// TIA Portal V16 export
// export: Created 2023-09-11T12:14:53.3184861Z, ExportSetting WithDefaults, DisplayName Totally Integrated Automation Portal, DisplayVersion V16 Update 6, DisplayName TIA Portal Version Control Interface, DisplayVersion V16 Update 2, DisplayName TIA Portal Openness, DisplayVersion V16 Update 6, DisplayName STEP 7 Professional, DisplayVersion V16 Update 6, DisplayName STEP 7 Safety, DisplayVersion V16, DisplayName WinCC Advanced, DisplayVersion V16 Update 6
FUNCTION "01_E_alarm handling" : Void   // FC10, LAD
TITLE = Boks Ready
{ S7_Optimized_Access := 'TRUE' }
AUTHOR : R.Tecmer
VERSION : 0.1
// Handling of alarms. Signaling and deleting
// stored: AutoNumber true, IsIECCheckEnabled false, SetENOAutomatically false, UDAEnableTagReadback false
   VAR_TEMP   // added for the SCL form of the ladder/FBD networks
      _w1 : Bool;
   END_VAR
BEGIN

REGION Network 1: Ready Inverters No1 No2
   // połączyłem bo usunięto drugi falownik
   // Jeśli brak gotowości to ustaw bity
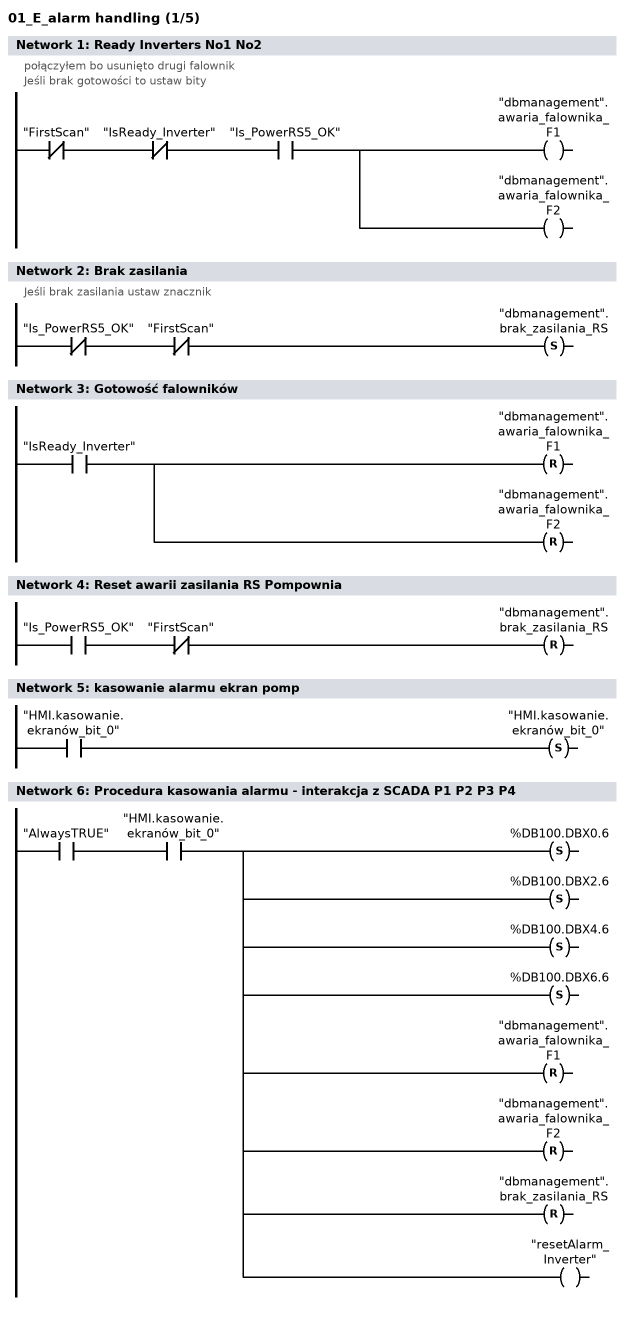
   RUNG wire#powerrail
      I_Contact( "FirstScan" )
      I_Contact( "IsReady_Inverter" )
      Contact( "Is_PowerRS5_OK" )
      wire#w1
      Coil( "dbmanagement".awaria_falownika_F1 )
   END_RUNG
   RUNG wire#w1
      Coil( "dbmanagement".awaria_falownika_F2 )
   END_RUNG
   // the same network as SCL:
   "dbmanagement".awaria_falownika_F1 := NOT "FirstScan" AND NOT "IsReady_Inverter" AND "Is_PowerRS5_OK";
   "dbmanagement".awaria_falownika_F2 := "dbmanagement".awaria_falownika_F1;
END_REGION

REGION Network 2: Brak zasilania
   // Jeśli brak zasilania ustaw znacznik
   RUNG wire#powerrail
      I_Contact( "Is_PowerRS5_OK" )
      I_Contact( "FirstScan" )
      S_Coil( "dbmanagement".brak_zasilania_RS )
   END_RUNG
   // the same network as SCL:
   IF NOT "Is_PowerRS5_OK" AND NOT "FirstScan" THEN "dbmanagement".brak_zasilania_RS := TRUE; END_IF;
END_REGION

REGION Network 3: Gotowość falowników
   RUNG wire#powerrail
      Contact( "IsReady_Inverter" )
      wire#w1
      R_Coil( "dbmanagement".awaria_falownika_F1 )
   END_RUNG
   RUNG wire#w1
      R_Coil( "dbmanagement".awaria_falownika_F2 )
   END_RUNG
   // the same network as SCL:
   IF "IsReady_Inverter" THEN
       "dbmanagement".awaria_falownika_F1 := FALSE;
       "dbmanagement".awaria_falownika_F2 := FALSE;
   END_IF;
END_REGION

REGION Network 4: Reset awarii zasilania RS Pompownia
   RUNG wire#powerrail
      Contact( "Is_PowerRS5_OK" )
      I_Contact( "FirstScan" )
      R_Coil( "dbmanagement".brak_zasilania_RS )
   END_RUNG
   // the same network as SCL:
   IF "Is_PowerRS5_OK" AND NOT "FirstScan" THEN "dbmanagement".brak_zasilania_RS := FALSE; END_IF;
END_REGION

REGION Network 5: kasowanie alarmu ekran pomp
   RUNG wire#powerrail
      Contact( "HMI.kasowanie.ekranów_bit_0" )
      S_Coil( "HMI.kasowanie.ekranów_bit_0" )
   END_RUNG
   // the same network as SCL:
   IF "HMI.kasowanie.ekranów_bit_0" THEN "HMI.kasowanie.ekranów_bit_0" := TRUE; END_IF;
END_REGION

REGION Network 6: Procedura kasowania alarmu - interakcja z SCADA P1 P2 P3 P4
   RUNG wire#powerrail
      Contact( "AlwaysTRUE" )
      Contact( "HMI.kasowanie.ekranów_bit_0" )
      wire#w1
      S_Coil( %DB100.DBX0.6 )
   END_RUNG
   RUNG wire#w1
      S_Coil( %DB100.DBX2.6 )
   END_RUNG
   RUNG wire#w1
      S_Coil( %DB100.DBX4.6 )
   END_RUNG
   RUNG wire#w1
      S_Coil( %DB100.DBX6.6 )
   END_RUNG
   RUNG wire#w1
      R_Coil( "dbmanagement".awaria_falownika_F1 )
   END_RUNG
   RUNG wire#w1
      R_Coil( "dbmanagement".awaria_falownika_F2 )
   END_RUNG
   RUNG wire#w1
      R_Coil( "dbmanagement".brak_zasilania_RS )
   END_RUNG
   RUNG wire#w1
      Coil( "resetAlarm_Inverter" )
   END_RUNG
   // the same network as SCL:
   #_w1 := "AlwaysTRUE" AND "HMI.kasowanie.ekranów_bit_0";
   IF #_w1 THEN
       %DB100.DBX0.6 := TRUE;
       %DB100.DBX2.6 := TRUE;
       %DB100.DBX4.6 := TRUE;
       %DB100.DBX6.6 := TRUE;
       "dbmanagement".awaria_falownika_F1 := FALSE;
       "dbmanagement".awaria_falownika_F2 := FALSE;
       "dbmanagement".brak_zasilania_RS := FALSE;
   END_IF;
   "resetAlarm_Inverter" := #_w1;
END_REGION

REGION Network 7: Reset błędu Soft-Start
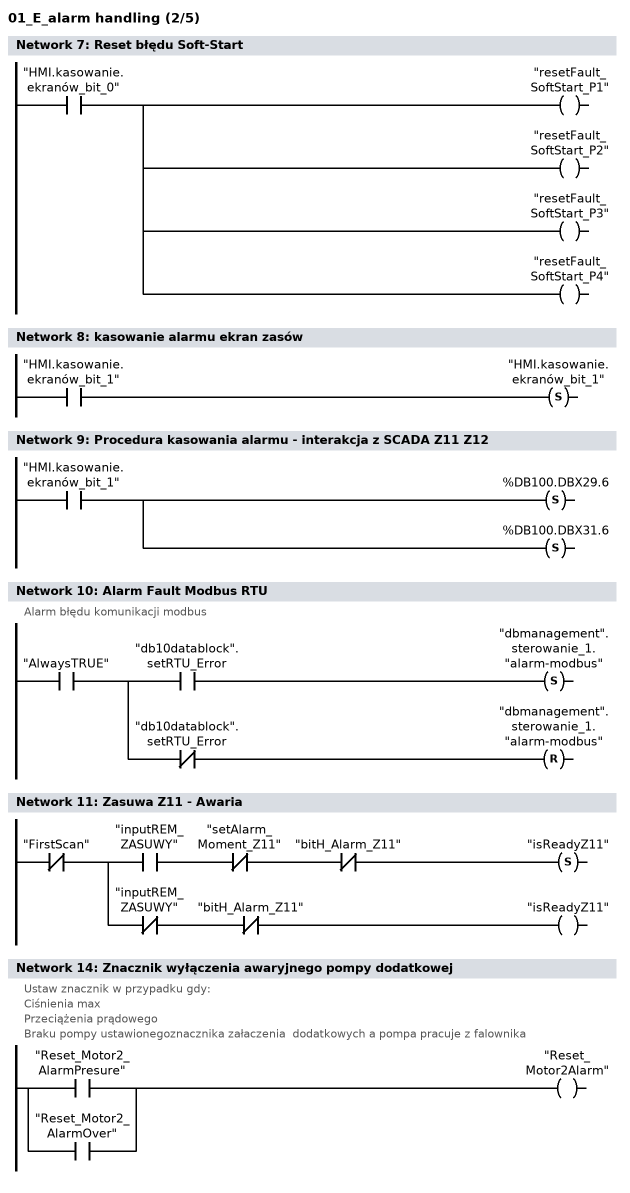
   RUNG wire#powerrail
      Contact( "HMI.kasowanie.ekranów_bit_0" )
      wire#w1
      Coil( "resetFault_SoftStart_P1" )
   END_RUNG
   RUNG wire#w1
      Coil( "resetFault_SoftStart_P2" )
   END_RUNG
   RUNG wire#w1
      Coil( "resetFault_SoftStart_P3" )
   END_RUNG
   RUNG wire#w1
      Coil( "resetFault_SoftStart_P4" )
   END_RUNG
   // the same network as SCL:
   "resetFault_SoftStart_P1" := "HMI.kasowanie.ekranów_bit_0";
   "resetFault_SoftStart_P2" := "HMI.kasowanie.ekranów_bit_0";
   "resetFault_SoftStart_P3" := "HMI.kasowanie.ekranów_bit_0";
   "resetFault_SoftStart_P4" := "HMI.kasowanie.ekranów_bit_0";
END_REGION

REGION Network 8: kasowanie alarmu ekran zasów
   RUNG wire#powerrail
      Contact( "HMI.kasowanie.ekranów_bit_1" )
      S_Coil( "HMI.kasowanie.ekranów_bit_1" )
   END_RUNG
   // the same network as SCL:
   IF "HMI.kasowanie.ekranów_bit_1" THEN "HMI.kasowanie.ekranów_bit_1" := TRUE; END_IF;
END_REGION

REGION Network 9: Procedura kasowania alarmu - interakcja z SCADA Z11 Z12
   RUNG wire#powerrail
      Contact( "HMI.kasowanie.ekranów_bit_1" )
      wire#w1
      S_Coil( %DB100.DBX29.6 )
   END_RUNG
   RUNG wire#w1
      S_Coil( %DB100.DBX31.6 )
   END_RUNG
   // the same network as SCL:
   IF "HMI.kasowanie.ekranów_bit_1" THEN
       %DB100.DBX29.6 := TRUE;
       %DB100.DBX31.6 := TRUE;
   END_IF;
END_REGION

REGION Network 10: Alarm Fault Modbus RTU
   // Alarm błędu komunikacji modbus
   RUNG wire#powerrail
      Contact( "AlwaysTRUE" )
      wire#w1
      Contact( "db10datablock".setRTU_Error )
      S_Coil( "dbmanagement".sterowanie_1."alarm-modbus" )
   END_RUNG
   RUNG wire#w1
      I_Contact( "db10datablock".setRTU_Error )
      R_Coil( "dbmanagement".sterowanie_1."alarm-modbus" )
   END_RUNG
   // the same network as SCL:
   IF "AlwaysTRUE" AND "db10datablock".setRTU_Error THEN
       "dbmanagement".sterowanie_1."alarm-modbus" := TRUE;
   END_IF;
   IF "AlwaysTRUE" AND NOT "db10datablock".setRTU_Error THEN
       "dbmanagement".sterowanie_1."alarm-modbus" := FALSE;
   END_IF;
END_REGION

REGION Network 11: Zasuwa Z11 - Awaria
   RUNG wire#powerrail
      I_Contact( "FirstScan" )
      wire#w1
      Contact( "inputREM_ZASUWY" )
      I_Contact( "setAlarm_Moment_Z11" )
      I_Contact( "bitH_Alarm_Z11" )
      S_Coil( "isReadyZ11" )
   END_RUNG
   RUNG wire#w1
      I_Contact( "inputREM_ZASUWY" )
      I_Contact( "bitH_Alarm_Z11" )
      Coil( "isReadyZ11" )
   END_RUNG
   // the same network as SCL:
   IF NOT "FirstScan" AND "inputREM_ZASUWY" AND NOT "setAlarm_Moment_Z11" AND NOT "bitH_Alarm_Z11" THEN
       "isReadyZ11" := TRUE;
   END_IF;
   "isReadyZ11" := NOT "FirstScan" AND NOT "inputREM_ZASUWY" AND NOT "bitH_Alarm_Z11";
END_REGION

REGION Network 12 (SCL): Z11 znacznik alarmu od momentówki w trybie zdalnym (aut/mamnual)
   IF  "inputAwariaMomentZ11" = False THEN
     // Ustaw alarm od momentu
     "setAlarm_Moment_Z11" := TRUE;
   ELSE
     "setAlarm_Moment_Z11" := FALSE;
     ;
   END_IF;
END_REGION

REGION Network 13 (SCL): Ustaw brak gotowości Z11
   IF "setAlarm_Moment_Z11" = TRUE OR "bitH_Alarm_Z11" THEN
     // Ustaw Alarm
     "isReadyZ11" := FALSE;

     ;
   END_IF;
END_REGION

REGION Network 14: Znacznik wyłączenia awaryjnego pompy dodatkowej
   // Ustaw znacznik w przypadku gdy:
   // Ciśnienia max
   // Przeciążenia prądowego
   // Braku pompy ustawionegoznacznika załaczenia  dodatkowych a pompa pracuje z falownika
   RUNG wire#powerrail
      Contact( "Reset_Motor2_AlarmPresure" )
      wire#w1
      Coil( "Reset_Motor2Alarm" )
   END_RUNG
   RUNG wire#powerrail
      Contact( "Reset_Motor2_AlarmOver" )
   END_RUNG wire#w1
   // the same network as SCL:
   "Reset_Motor2Alarm" := "Reset_Motor2_AlarmPresure" OR "Reset_Motor2_AlarmOver";
END_REGION

REGION Network 15: Znacznik wyłączenia awaryjnego pompy dodatkowej
   // Ustawienie w przypadku:
   // Ciśnienia max
   // Przeciążenia prądowego
   // Braku pompy dodatkowych
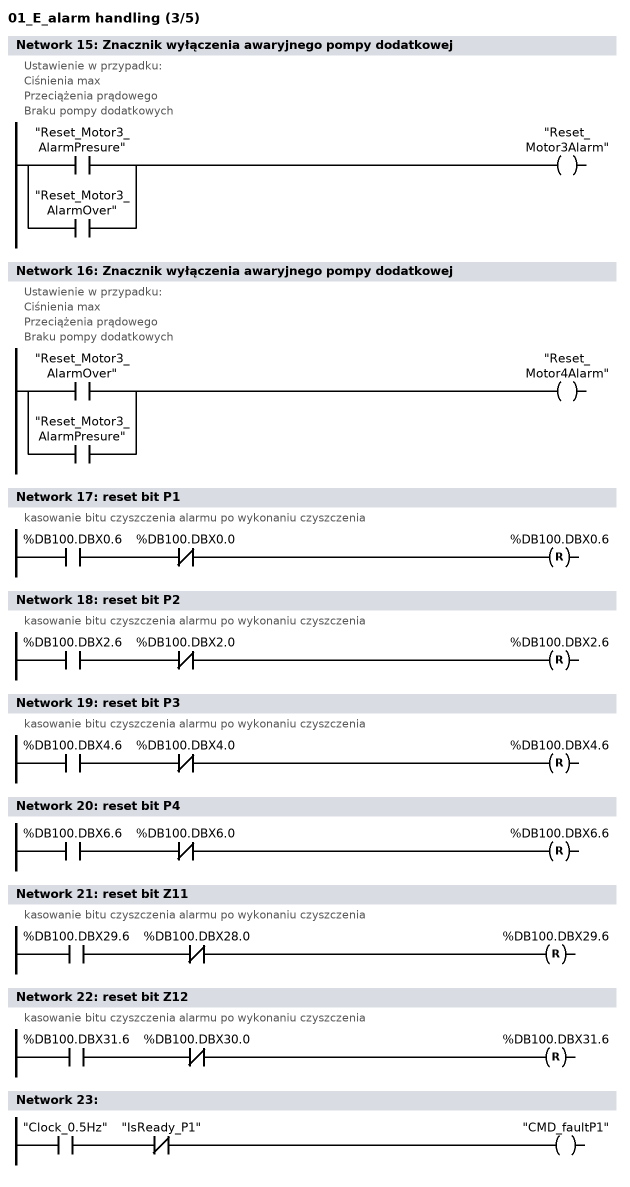
   RUNG wire#powerrail
      Contact( "Reset_Motor3_AlarmPresure" )
      wire#w1
      Coil( "Reset_Motor3Alarm" )
   END_RUNG
   RUNG wire#powerrail
      Contact( "Reset_Motor3_AlarmOver" )
   END_RUNG wire#w1
   // the same network as SCL:
   "Reset_Motor3Alarm" := "Reset_Motor3_AlarmPresure" OR "Reset_Motor3_AlarmOver";
END_REGION

REGION Network 16: Znacznik wyłączenia awaryjnego pompy dodatkowej
   // Ustawienie w przypadku:
   // Ciśnienia max
   // Przeciążenia prądowego
   // Braku pompy dodatkowych
   RUNG wire#powerrail
      Contact( "Reset_Motor3_AlarmOver" )
      wire#w1
      Coil( "Reset_Motor4Alarm" )
   END_RUNG
   RUNG wire#powerrail
      Contact( "Reset_Motor3_AlarmPresure" )
   END_RUNG wire#w1
   // the same network as SCL:
   "Reset_Motor4Alarm" := "Reset_Motor3_AlarmOver" OR "Reset_Motor3_AlarmPresure";
END_REGION

REGION Network 17: reset bit P1
   // kasowanie bitu czyszczenia alarmu po wykonaniu czyszczenia
   RUNG wire#powerrail
      Contact( %DB100.DBX0.6 )
      I_Contact( %DB100.DBX0.0 )
      R_Coil( %DB100.DBX0.6 )
   END_RUNG
   // the same network as SCL:
   IF %DB100.DBX0.6 AND NOT %DB100.DBX0.0 THEN %DB100.DBX0.6 := FALSE; END_IF;
END_REGION

REGION Network 18: reset bit P2
   // kasowanie bitu czyszczenia alarmu po wykonaniu czyszczenia
   RUNG wire#powerrail
      Contact( %DB100.DBX2.6 )
      I_Contact( %DB100.DBX2.0 )
      R_Coil( %DB100.DBX2.6 )
   END_RUNG
   // the same network as SCL:
   IF %DB100.DBX2.6 AND NOT %DB100.DBX2.0 THEN %DB100.DBX2.6 := FALSE; END_IF;
END_REGION

REGION Network 19: reset bit P3
   // kasowanie bitu czyszczenia alarmu po wykonaniu czyszczenia
   RUNG wire#powerrail
      Contact( %DB100.DBX4.6 )
      I_Contact( %DB100.DBX4.0 )
      R_Coil( %DB100.DBX4.6 )
   END_RUNG
   // the same network as SCL:
   IF %DB100.DBX4.6 AND NOT %DB100.DBX4.0 THEN %DB100.DBX4.6 := FALSE; END_IF;
END_REGION

REGION Network 20: reset bit P4
   RUNG wire#powerrail
      Contact( %DB100.DBX6.6 )
      I_Contact( %DB100.DBX6.0 )
      R_Coil( %DB100.DBX6.6 )
   END_RUNG
   // the same network as SCL:
   IF %DB100.DBX6.6 AND NOT %DB100.DBX6.0 THEN %DB100.DBX6.6 := FALSE; END_IF;
END_REGION

REGION Network 21: reset bit Z11
   // kasowanie bitu czyszczenia alarmu po wykonaniu czyszczenia
   RUNG wire#powerrail
      Contact( %DB100.DBX29.6 )
      I_Contact( %DB100.DBX28.0 )
      R_Coil( %DB100.DBX29.6 )
   END_RUNG
   // the same network as SCL:
   IF %DB100.DBX29.6 AND NOT %DB100.DBX28.0 THEN %DB100.DBX29.6 := FALSE; END_IF;
END_REGION

REGION Network 22: reset bit Z12
   // kasowanie bitu czyszczenia alarmu po wykonaniu czyszczenia
   RUNG wire#powerrail
      Contact( %DB100.DBX31.6 )
      I_Contact( %DB100.DBX30.0 )
      R_Coil( %DB100.DBX31.6 )
   END_RUNG
   // the same network as SCL:
   IF %DB100.DBX31.6 AND NOT %DB100.DBX30.0 THEN %DB100.DBX31.6 := FALSE; END_IF;
END_REGION

REGION Network 23
   RUNG wire#powerrail
      Contact( "Clock_0.5Hz" )
      I_Contact( "IsReady_P1" )
      Coil( "CMD_faultP1" )
   END_RUNG
   // the same network as SCL:
   "CMD_faultP1" := "Clock_0.5Hz" AND NOT "IsReady_P1";
END_REGION

REGION Network 24
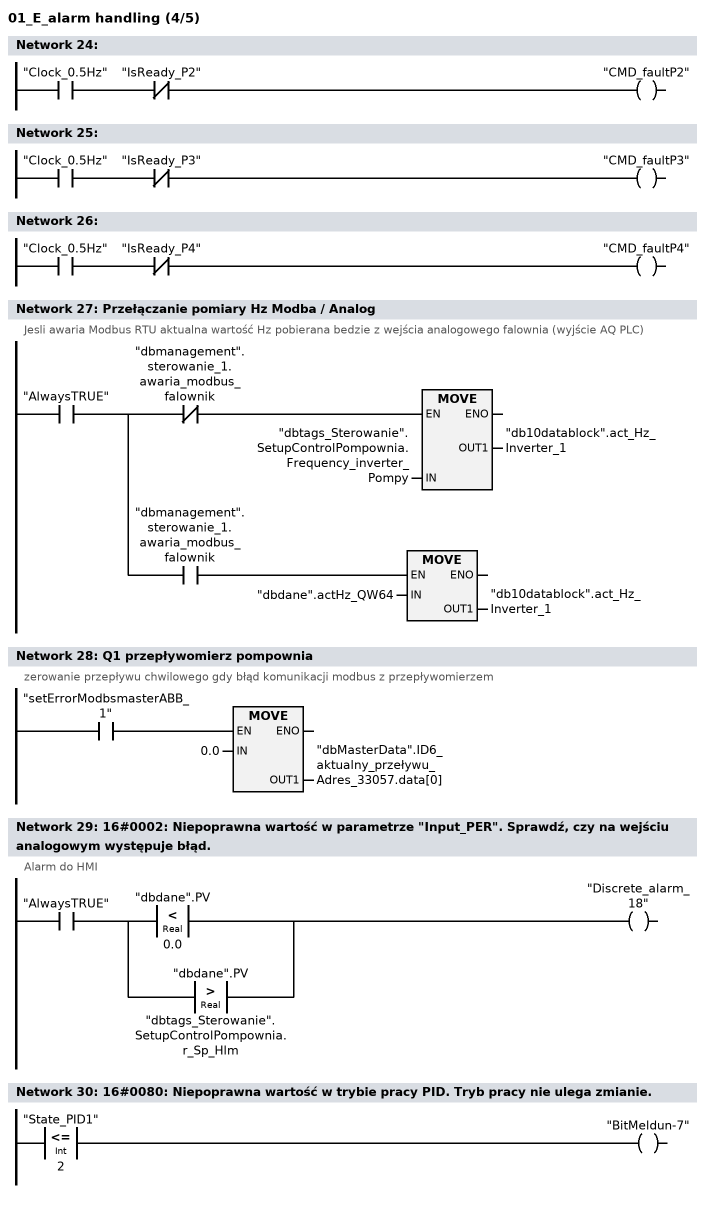
   RUNG wire#powerrail
      Contact( "Clock_0.5Hz" )
      I_Contact( "IsReady_P2" )
      Coil( "CMD_faultP2" )
   END_RUNG
   // the same network as SCL:
   "CMD_faultP2" := "Clock_0.5Hz" AND NOT "IsReady_P2";
END_REGION

REGION Network 25
   RUNG wire#powerrail
      Contact( "Clock_0.5Hz" )
      I_Contact( "IsReady_P3" )
      Coil( "CMD_faultP3" )
   END_RUNG
   // the same network as SCL:
   "CMD_faultP3" := "Clock_0.5Hz" AND NOT "IsReady_P3";
END_REGION

REGION Network 26
   RUNG wire#powerrail
      Contact( "Clock_0.5Hz" )
      I_Contact( "IsReady_P4" )
      Coil( "CMD_faultP4" )
   END_RUNG
   // the same network as SCL:
   "CMD_faultP4" := "Clock_0.5Hz" AND NOT "IsReady_P4";
END_REGION

REGION Network 27: Przełączanie pomiary Hz Modba / Analog
   // Jesli awaria Modbus RTU aktualna wartość Hz pobierana bedzie z wejścia analogowego falownia (wyjście AQ PLC)
   RUNG wire#powerrail
      Contact( "AlwaysTRUE" )
      wire#w1
      I_Contact( "dbmanagement".sterowanie_1.awaria_modbus_falownik )
      Move(in := "dbtags_Sterowanie".SetupControlPompownia.Frequency_inverter_Pompy, out1 => "db10datablock".act_Hz_Inverter_1)
   END_RUNG
   RUNG wire#w1
      Contact( "dbmanagement".sterowanie_1.awaria_modbus_falownik )
      Move(in := "dbdane".actHz_QW64, out1 => "db10datablock".act_Hz_Inverter_1)
   END_RUNG
   // the same network as SCL:
   IF "AlwaysTRUE" AND NOT "dbmanagement".sterowanie_1.awaria_modbus_falownik THEN
       "db10datablock".act_Hz_Inverter_1 := "dbtags_Sterowanie".SetupControlPompownia.Frequency_inverter_Pompy;
   END_IF;
   IF "AlwaysTRUE" AND "dbmanagement".sterowanie_1.awaria_modbus_falownik THEN
       "db10datablock".act_Hz_Inverter_1 := "dbdane".actHz_QW64;
   END_IF;
END_REGION

REGION Network 28: Q1 przepływomierz pompownia
   // zerowanie przepływu chwilowego gdy błąd komunikacji modbus z przepływomierzem
   RUNG wire#powerrail
      Contact( "setErrorModbsmasterABB_1" )
      { S7_GenerateENO := "TRUE" } Move(in := 0.0, out1 => "dbMasterData".ID6_aktualny_przeływu_Adres_33057.data[0])
   END_RUNG
   // the same network as SCL:
   IF "setErrorModbsmasterABB_1" THEN
       "dbMasterData".ID6_aktualny_przeływu_Adres_33057.data[0] := 0.0;
   END_IF;
END_REGION

REGION Network 29: 16#0002: Niepoprawna wartość w parametrze "Input_PER". Sprawdź, czy na wejściu analogowym występuje błąd.
   // Alarm do HMI
   RUNG wire#powerrail
      Contact( "AlwaysTRUE" )
      wire#w1
      { S7_Templates := "SrcType := Real" } LT_Contact(in1 := "dbdane".PV, in2 := 0.0)
      wire#w2
      Coil( "Discrete_alarm_18" )
   END_RUNG
   RUNG wire#w1
      { S7_Templates := "SrcType := Real" } GT_Contact(in1 := "dbdane".PV, in2 := "dbtags_Sterowanie".SetupControlPompownia.r_Sp_Hlm)
   END_RUNG wire#w2
   // the same network as SCL:
   "Discrete_alarm_18" := "AlwaysTRUE" AND (("dbdane".PV < 0.0) OR ("dbdane".PV > "dbtags_Sterowanie".SetupControlPompownia.r_Sp_Hlm));
END_REGION

REGION Network 30: 16#0080: Niepoprawna wartość w trybie pracy PID. Tryb pracy nie ulega zmianie.
   RUNG wire#powerrail
      { S7_Templates := "SrcType := Int" } LE_Contact(in1 := "State_PID1", in2 := 2)
      Coil( "BitMeldun-7" )
   END_RUNG
   // the same network as SCL:
   "BitMeldun-7" := "State_PID1" <= 2;
END_REGION

REGION Network 31: 16#1000: Niepoprawna wartość w parametrze "Wartość zadana": Wartość nie ma prawidłowego formatu liczbowego.
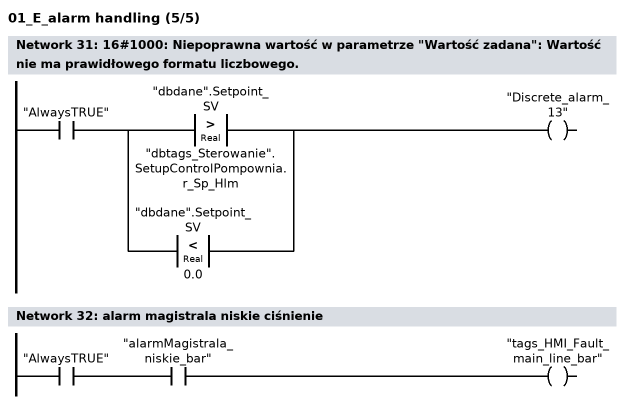
   RUNG wire#powerrail
      Contact( "AlwaysTRUE" )
      wire#w1
      { S7_Templates := "SrcType := Real" } GT_Contact(in1 := "dbdane".Setpoint_SV, in2 := "dbtags_Sterowanie".SetupControlPompownia.r_Sp_Hlm)
      wire#w2
      Coil( "Discrete_alarm_13" )
   END_RUNG
   RUNG wire#w1
      { S7_Templates := "SrcType := Real" } LT_Contact(in1 := "dbdane".Setpoint_SV, in2 := 0.0)
   END_RUNG wire#w2
   // the same network as SCL:
   "Discrete_alarm_13" := "AlwaysTRUE" AND (("dbdane".Setpoint_SV > "dbtags_Sterowanie".SetupControlPompownia.r_Sp_Hlm) OR ("dbdane".Setpoint_SV < 0.0));
END_REGION

REGION Network 32: alarm magistrala niskie ciśnienie
   RUNG wire#powerrail
      Contact( "AlwaysTRUE" )
      Contact( "alarmMagistrala_niskie_bar" )
      Coil( "tags_HMI_Fault_main_line_bar" )
   END_RUNG
   // the same network as SCL:
   "tags_HMI_Fault_main_line_bar" := "AlwaysTRUE" AND "alarmMagistrala_niskie_bar";
END_REGION
END_FUNCTION
